{attribute addProperty BoxType "KL9900-0054"}
{attribute addProperty Id "Channel_1Channel_6514201C00"}
{attribute addProperty CRC "2994480759"}
{attribute addProperty SizeInBites "0"}
{attribute addProperty SizeInBytes "0"}
TYPE KL_B27C2677 :
STRUCT
	{attribute addProperty Name "Channel_1"}
	Channel_1 : Channel_6514201C;
END_STRUCT
END_TYPE

(* stored: Version 1.2.0.0, ProductVersion 3.1.4024.9
   DUT KL_B27C2677: Id {393128f8-030f-43ca-95a3-97f960e09a43} *)
